// TIA Portal V20 export
// export: Created 2026-04-11T06:02:30.4089393Z, ExportSetting WithDefaults, DisplayName Totally Integrated Automation Portal, DisplayVersion V20, DisplayName TIA Portal Openness, DisplayVersion V20, DisplayName TIA Portal Version Control Interface, DisplayVersion V20, DisplayName STEP 7 Professional, DisplayVersion V20, DisplayName STEP 7 Safety, DisplayVersion V20, DisplayName WinCC Basic/Comfort/Advanced, DisplayVersion V20, DisplayName WinCC Unified, DisplayVersion V20
TYPE "udtHMI_PID_Compact"
// stored: IsFailsafeCompliant false
   STRUCT
      iMode : Int;   // Current mode
      iPIDMode { ExternalWritable := 'False'} : Int;   // PID compact mode
      iErrorCode { ExternalWritable := 'False'} : Int;   // Error code
      iEstopFunction { S7_SetPoint := 'True'} : Int;   // Enum of E-Stop repsonse (Estop.xxx)
      rEstopOverride { S7_SetPoint := 'True'} : Real;   // PID output value for an e-stop if custom value is selected
      rManualOverride { S7_SetPoint := 'True'} : Real;   // PID output value for an operator override
      rAutoOverride { ExternalWritable := 'False'} : Real;   // PID output value for a PLC override
      rManualSP { S7_SetPoint := 'True'} : Real;   // PID set point for manual mode
      rAutoSP { ExternalWritable := 'False'} : Real;   // PID set point for automatic mode
      rActualInput { ExternalWritable := 'False'} : Real;   // Actual PID input value
      wActualInputPeripheral { ExternalWritable := 'False'} : Word;   // Actual PID input peripheral value
      rOutput { ExternalWritable := 'False'} : Real;   // PID output value
      wOutputPeripheral { ExternalWritable := 'False'} : Word;   // PID output peripheral value
      bOutputPWM { ExternalWritable := 'False'} : Bool;   // PID output value for PWM
      rProportionalGain { S7_SetPoint := 'True'} : Real;   // Proportional gain coefficient
      rIntegralTime { S7_SetPoint := 'True'} : Real;   // Integral control time
      rDerivativeTime { S7_SetPoint := 'True'} : Real;   // Derivative control time
      rProportionalWeight { S7_SetPoint := 'True'} : Real;   // Proportional control weighting
      rDerivativeWeight { S7_SetPoint := 'True'} : Real;   // Derivative control weighting
      bPB_ResetError : Bool;   // PB Reset errors
      bPB_Pretune : Bool;   // PB Start pretuning
      bPB_FineTune : Bool;   // PB Start finetuning
      bPB_AutomaticMode : Bool;   // PB Switch to automatic mode
      bPB_ManualMode : Bool;   // PB Switch to manual mode
      bPB_ManualTuning : Bool;   // PB Switch to manual PID tuning
      bTOG_ManualTuning { ExternalWritable := 'False'} : Bool;   // TOG Manual tuning enabled
      bPBEN_ResetError { ExternalWritable := 'False'} : Bool;   // PB Reset errors enabled
      bPBEN_Pretune { ExternalWritable := 'False'} : Bool;   // PB Pretuning enabled
      bPBEN_FineTune { ExternalWritable := 'False'} : Bool;   // PB Fine tuning enabled
      bPBEN_AutomaticMode { ExternalWritable := 'False'} : Bool;   // PB Automatic mode enabled
      bPBEN_ManualMode { ExternalWritable := 'False'} : Bool;   // PB Manual mode enabled
      bError { ExternalWritable := 'False'} : Bool;   // Overall error
   END_STRUCT;
END_TYPE
